TYPE "PPrf_Pivot"
VERSION : 0.1
// Block: PPrf_Pivot
   STRUCT
      PrgNo : DInt;
      PrgName : "String[79]";
      RecordNo : Int;
   END_STRUCT;

END_TYPE
